Staubli VAL3: stringtopoint.pgx

program stringtopoint(string x_sString (dimensions=1), num x_nNum (dimensions=1))
  local string l_s
  local bool l_btest
  local num nX
  local num nY
  local num nZ
  local num nA
  local num nB
  local num nC
  local pointRx l_pPointRx
  local trsf tTrsf
  local pointRx pChangeMid1
  local num nP
  local pointRx pChangeMid2
begin
  l_s=x_sString
  l_s=toNum(l_s,nX,l_btest)
  l_s=toNum(l_s,nY,l_btest)
  l_s=toNum(l_s,nZ,l_btest)
  l_s=toNum(l_s,nA,l_btest)
  l_s=toNum(l_s,nB,l_btest)
  l_s=toNum(l_s,nC,l_btest)
  l_s=toNum(l_s,nP,l_btest)
  nPulse[x_nNum]=nP
  pChange.trsf.x=nX
  pChange.trsf.z=nZ
  pChange.trsf.y=nY
  ////  pChangeMid=compose(pChange,FrmDraw,{0,0,0,0,90,0})
  ////  pfrmCad[x_nNum]=compose(pChangeMid,FrmDraw,{0,0,0,0,0,nC})
  pChangeMid1=compose(pChange,FrmDraw,{0,0,0,nA,0,0})
  pChangeMid2=compose(pChangeMid1,FrmDraw,{0,0,0,0,0,nB})
  pfrmCad[x_nNum]=compose(pChangeMid2,FrmDraw,{0,0,0,nC,0,0})
  pfrmCad[x_nNum].trsf.x=pChange.trsf.x
  pfrmCad[x_nNum].trsf.z=pChange.trsf.z
  pfrmCad[x_nNum].trsf.y=pChange.trsf.y
  pChange[0].trsf={0,0,0,0,0,0}
end
